PROGRAM MAIN
VAR
	bSendMessagePDF	: BOOL;
	bSendMessageMP4	: BOOL;
	
	bIsInitalized 	: BOOL;
	
	fbMessagePDF	: FB_TcMessage;	
	fbMessageMP4	: FB_TcMessage;
	
	hr 				: HRESULT;
	hrLastError 	: HRESULT;
END_VAR


// init
IF NOT bIsInitalized THEN	
	bIsInitalized := TRUE;	
	hr := fbMessagePDF.CreateEx(TC_EVENTS.TestEvents.Event_PDF, 0);
	hr := fbMessageMP4.CreateEx(TC_EVENTS.TestEvents.Event_MP4, 0);
END_IF

// send message for pdf user guidance
IF bSendMessagePDF THEN
	bSendMessagePDF := FALSE;
	hr := fbMessagePDF.Send(0);
END_IF
// send message for mp4 user guidance
IF bSendMessageMP4 THEN
	bSendMessageMP4 := FALSE;
	hr := fbMessageMP4.Send(0);
END_IF

// error feedback
IF FAILED(hr) THEN
	hrLastError := hr;
END_IF

END_PROGRAM

(* stored: Version 1.1.0.1
   POU MAIN: Id {f6e84080-761d-4928-b350-ecd69bc0a128}, SpecialFunc None *)
